# EPICS substitutions: viocs/ts_ps/ts_psApp/Db/quad.substitutions
file "db/individual.db" {
    pattern { family, pos }
        { "QF", "01-A"}
        { "QF", "01-B"}
        { "QD", "02"}
        { "QF", "02"}
        { "QF", "03"}
        { "QD", "04-A"}
        { "QF", "04"}
        { "QD", "04-B"}
}
